// TIA Portal project "P7" (V17)

(* hardware
DEVICE "S7-1500/ET200MP station_1"  S7-1500 station
   slot 0: "Rail_0"  Rack  6ES7 590-1***0-0AA0
   slot 1: "PLC_1"  CPU 1515-2 PN  6ES7 515-2AM02-0AB0  V2.9
      slot 3: "CPU display_1"  6ES7591-1BA00-0AA0
      slot 32768: "PROFINET interface_1"  X1
         slot 32769: "Port_1"  X1 P1
         slot 32770: "Port_2"  X1 P2
      slot 33024: "PROFINET interface_2"  X2
         slot 33025: "Port_1"  X2 P1
      slot 34817: "Virtual CP interface port_1"  Virtual CP interface port  Virtual CP interface port
*)

// ===== PLC "PLC_1"  CPU 1515-2 PN =====

VAR_GLOBAL   // PLC tag table "Default tag table"
   "SET PRESSURE" AT %MD500 : Real;
   "ACTUAL PRESSURE" AT %MD704 : Real;
   "4-20 mA FROM PT OUTPUT" AT %IW96 : Int;
   "Manual Mode Enable" AT %M61.1 : Bool;
   "PID CONTROLLER RESET" AT %M61.2 : Bool;
   "PID OUTPUT" AT %MD758 : Real;
   "PID OUTPUT ANALOG" AT %MW762 : Int;
   "PID HIGH LIMIT" AT %M766.0 : Bool;
   "PID LOW LIMIT" AT %M766.1 : Bool;
   "PID INPUT WARNING" AT %M766.2 : Bool;
   "PID STATE WORD" AT %MW770 : Int;
   "PID ERROR WORD" AT %M778.0 : Bool;
   "RUN MODE BY START UP" AT %M0.3 : Bool;
   "INLET VALVE FOR REACTANTS" AT %QW96 : Int;
   "OUTLET VALVE FOR PRODUCTS" AT %QW98 : Int;
END_VAR

ORGANIZATION_BLOCK "Main"   // OB1, LAD, ProgramCycle
TITLE = "Main Program Sweep (Cycle)"
{ S7_Optimized_Access := 'TRUE' }
VERSION : 0.1
   VAR_INPUT
      Initial_Call : Bool;   // Initial call of this OB
      Remanence : Bool;   // =True, if remanent data are available
   END_VAR
BEGIN

REGION Network 1: Integral Action Time (Ti) Proporcional Gain
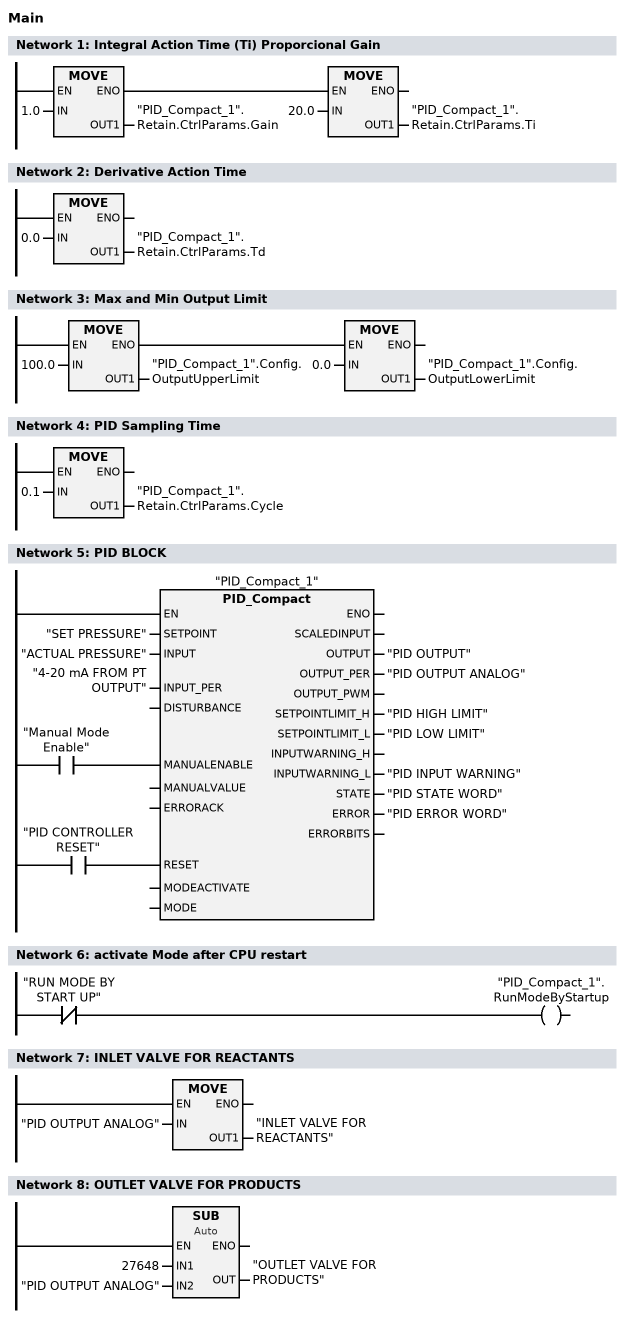
   RUNG wire#powerrail
      Move(in := 1.0, out1 => "PID_Compact_1".Retain.CtrlParams.Gain)
      Move(in := 20.0, out1 => "PID_Compact_1".Retain.CtrlParams.Ti)
   END_RUNG
   // the same network as SCL:
   "PID_Compact_1".Retain.CtrlParams.Gain := 1.0;
   "PID_Compact_1".Retain.CtrlParams.Ti := 20.0;
END_REGION

REGION Network 2: Derivative Action Time
   RUNG wire#powerrail
      Move(in := 0.0, out1 => "PID_Compact_1".Retain.CtrlParams.Td)
   END_RUNG
   // the same network as SCL:
   "PID_Compact_1".Retain.CtrlParams.Td := 0.0;
END_REGION

REGION Network 3: Max and Min Output Limit
   RUNG wire#powerrail
      Move(in := 100.0, out1 => "PID_Compact_1".Config.OutputUpperLimit)
      Move(in := 0.0, out1 => "PID_Compact_1".Config.OutputLowerLimit)
   END_RUNG
   // the same network as SCL:
   "PID_Compact_1".Config.OutputUpperLimit := 100.0;
   "PID_Compact_1".Config.OutputLowerLimit := 0.0;
END_REGION

REGION Network 4: PID Sampling Time
   RUNG wire#powerrail
      Move(in := 0.1, out1 => "PID_Compact_1".Retain.CtrlParams.Cycle)
   END_RUNG
   // the same network as SCL:
   "PID_Compact_1".Retain.CtrlParams.Cycle := 0.1;
END_REGION

REGION Network 5: PID BLOCK
   "PID_Compact_1"(Setpoint := "SET PRESSURE",   // PID_Compact
                   Input := "ACTUAL PRESSURE",
                   Input_PER := "4-20 mA FROM PT OUTPUT",
                   ManualEnable := "Manual Mode Enable",
                   Reset := "PID CONTROLLER RESET",
                   Output => "PID OUTPUT",
                   Output_PER => "PID OUTPUT ANALOG",
                   SetpointLimit_H => "PID HIGH LIMIT",
                   SetpointLimit_L => "PID LOW LIMIT",
                   InputWarning_L => "PID INPUT WARNING",
                   State => "PID STATE WORD",
                   Error => "PID ERROR WORD");
END_REGION

REGION Network 6: activate Mode after CPU restart
   RUNG wire#powerrail
      I_Contact( "RUN MODE BY START UP" )
      Coil( "PID_Compact_1".RunModeByStartup )
   END_RUNG
   // the same network as SCL:
   "PID_Compact_1".RunModeByStartup := NOT "RUN MODE BY START UP";
END_REGION

REGION Network 7: INLET VALVE FOR REACTANTS
   RUNG wire#powerrail
      Move(in := "PID OUTPUT ANALOG", out1 => "INLET VALVE FOR REACTANTS")
   END_RUNG
   // the same network as SCL:
   "INLET VALVE FOR REACTANTS" := "PID OUTPUT ANALOG";
END_REGION

REGION Network 8: OUTLET VALVE FOR PRODUCTS
   RUNG wire#powerrail
      Sub(in1 := 27648, in2 := "PID OUTPUT ANALOG", out => "OUTLET VALVE FOR PRODUCTS")
   END_RUNG
   // the same network as SCL:
   "OUTLET VALVE FOR PRODUCTS" := 27648 - "PID OUTPUT ANALOG";
END_REGION
END_ORGANIZATION_BLOCK